// TwinCAT 3 PLC project Test_Proj
// ProgramVersion: 3.1.4026.13
// libraries:
//   Tc2_MC2, * (Beckhoff Automation GmbH)
//   Tc2_Standard, * (Beckhoff Automation GmbH)
//   Tc2_System, * (Beckhoff Automation GmbH)
//   Tc3PlcTestSuite, * (Simmel)
//   [Motion Library], * (Beckhoff UK)
// project tree:
//   / PlcTask.TcTTO
//   POUs/ AxisPowerTestSuite.TcPOU, AxisResetTestSuite.TcPOU, MAIN.TcPOU
// real-time tasks:
//   TASK PlcTask: cycle T#10ms, priority 20, ADS port 350

CONFIGURATION Test_Proj
    RESOURCE PLC ON TwinCAT3
        TASK PlcTask(INTERVAL := T#10ms, PRIORITY := 20);
        PROGRAM MAIN WITH PlcTask : MAIN;
    END_RESOURCE
END_CONFIGURATION

// ---- POUs/MAIN.TcPOU
PROGRAM MAIN
VAR
	PowerTestSuite : AxisPowerTestSuite;
	ResetTestSuite : AxisResetTestSuite;
END_VAR

PowerTestSuite();
ResetTestSuite();

END_PROGRAM

// ---- POUs/AxisPowerTestSuite.TcPOU
FUNCTION_BLOCK AxisPowerTestSuite
VAR
	StubAxis : AXIS_REF;
	TestAxisPower : AxisPower(StubAxis);
	ReRun: BOOL;
END_VAR

DoesAxisAcceptEnable_Test();
RejectEnableWhenEnabled_Test();
IF ReRun THEN
	TestSuite.ReRunTests();
	ReRun := FALSE;
END_IF

METHOD DoesAxisAcceptEnable_Test : BOOL
VAR_INST
	Expected : HRESULT;
	Actual	 : HRESULT;
END_VAR
IF TestSuite.Test(__POUNAME()).ExecuteTest() THEN
	Expected := s_OK;
	Actual := TestAxisPower.Enable();
	TestAxisPower.Disable();
	TestSuite.Test(__POUNAME()).AssertEqual(Expected, Actual);
END_IF
END_METHOD

METHOD RejectEnableWhenEnabled_Test : BOOL
VAR_INST
	Expected : HRESULT;
	Actual	 : HRESULT;
END_VAR
IF TestSuite.Test(__POUNAME()).ExecuteTest() THEN
	Expected := s_OK;
	TestAxisPower.Enable();
	Actual := TestAxisPower.Enable();
	TestAxisPower.Disable();
	TestSuite.Test(__POUNAME()).AssertEqual(Expected, Actual);
END_IF
END_METHOD

END_FUNCTION_BLOCK

// ---- POUs/AxisResetTestSuite.TcPOU
FUNCTION_BLOCK AxisResetTestSuite
VAR
	_axis : AXIS_REF;
	TestAxisReset : AxesReset(_axis);
	ReRun: BOOL;
END_VAR

DoesAcceptExecute_Test();
RejectResetWhileResetting_Test();
IF ReRun THEN
	TestSuite.ReRunTests();
	ReRun := FALSE;
END_IF

METHOD DoesAcceptExecute_Test : BOOL
VAR_INST
	Expected : HRESULT;
	Actual	 : HRESULT;
END_VAR
IF TestSuite.Test(__POUNAME()).ExecuteTest() THEN
	Expected := s_OK;
	Actual := TestAxisReset.Execute();
	TestAxisReset.Abort();
	TestSuite.Test(__POUNAME()).AssertEqual(Expected, Actual);
END_IF
END_METHOD

METHOD RejectResetWhileResetting_Test : BOOL
VAR_INST
	Expected : HRESULT;
	Actual	 : HRESULT;
END_VAR
IF TestSuite.Test(__POUNAME()).ExecuteTest() THEN
	Expected := S_FALSE;
	TestAxisReset.Execute();
	Actual := TestAxisReset.Execute();
	TestSuite.Test(__POUNAME()).AssertEqual(Expected, Actual);
END_IF
END_METHOD

END_FUNCTION_BLOCK
